// TIA Portal V17 export
// export: Created 2024-08-26T21:07:16.3751561Z, ExportSetting WithDefaults, DisplayName Totally Integrated Automation Portal, DisplayVersion V17 Update 7, DisplayName TIA Portal Openness, DisplayVersion V17 Update 7, DisplayName TIA Portal Version Control Interface, DisplayVersion V17, DisplayName SINAMICS Startdrive Advanced, DisplayVersion V17 SP2, DisplayName SINAMICS Startdrive G110M, G120, G120C, G120D, G120P, G115D, DisplayVersion V17 SP2, DisplayName SINAMICS Startdrive G130, G150, S120, S150, SINAMICS MV, S210, DisplayVersion V17 SP2, DisplayName STEP 7 Professional, DisplayVersion V17 Update 7, DisplayName STEP 7 Safety, DisplayVersion V17 Update 6, DisplayName WinCC Advanced / Unified PC, DisplayVersion V17 Update 7
FUNCTION "cylinderControl" : Void   // FC9, LAD
{ S7_Optimized_Access := 'TRUE' }
VERSION : 0.1
// stored: AutoNumber true, IsIECCheckEnabled false, SetENOAutomatically false, UDAEnableTagReadback false
   VAR_TEMP
      enableCylinders : Bool;
   END_VAR
   VAR_TEMP   // added for the SCL form of the ladder/FBD networks
      _w1 : Bool;
      _w2 : Bool;
   END_VAR
BEGIN

REGION Network 1
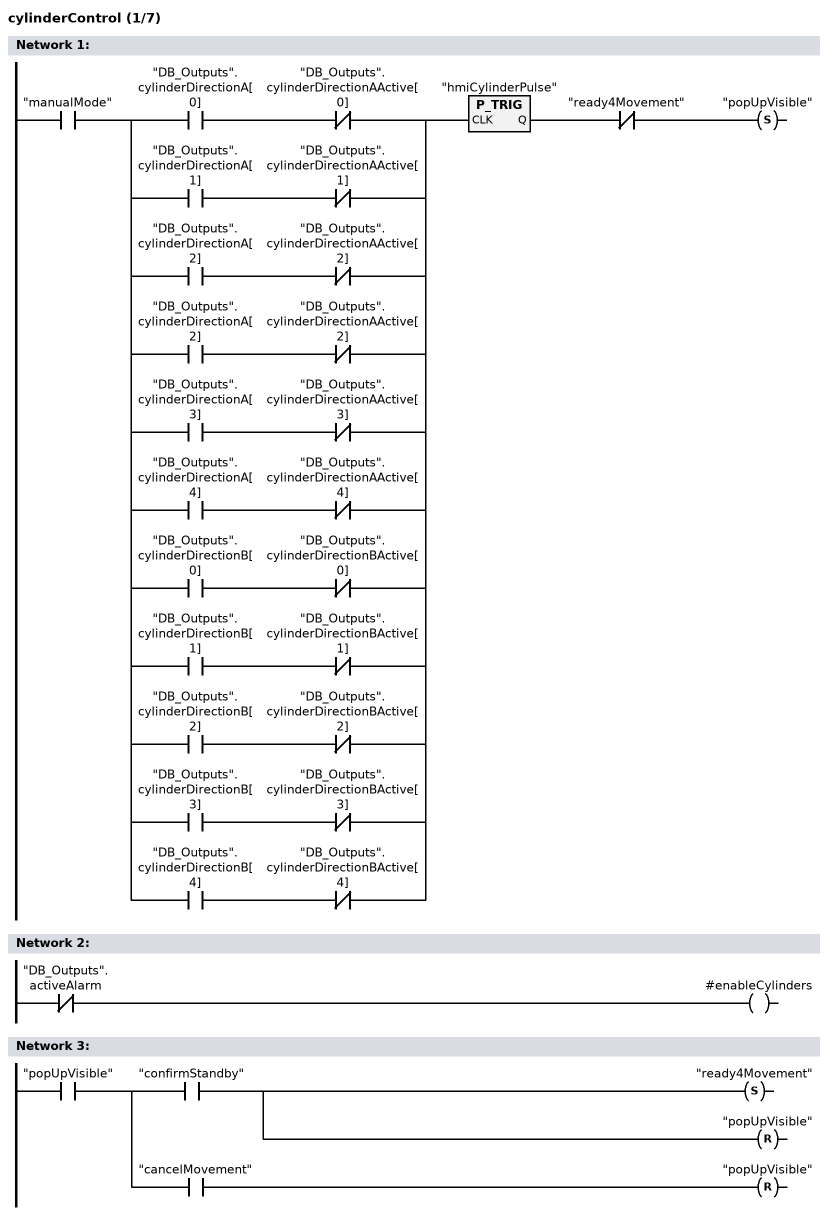
   RUNG wire#powerrail
      Contact( "manualMode" )
      wire#w1
      Contact( "DB_Outputs".cylinderDirectionA[0] )
      I_Contact( "DB_Outputs".cylinderDirectionAActive[0] )
      wire#w2
      P_Trig( "hmiCylinderPulse" )
      I_Contact( "ready4Movement" )
      S_Coil( "popUpVisible" )
   END_RUNG
   RUNG wire#w1
      Contact( "DB_Outputs".cylinderDirectionA[1] )
      I_Contact( "DB_Outputs".cylinderDirectionAActive[1] )
   END_RUNG wire#w2
   RUNG wire#w1
      Contact( "DB_Outputs".cylinderDirectionA[2] )
      I_Contact( "DB_Outputs".cylinderDirectionAActive[2] )
   END_RUNG wire#w2
   RUNG wire#w1
      Contact( "DB_Outputs".cylinderDirectionA[2] )
      I_Contact( "DB_Outputs".cylinderDirectionAActive[2] )
   END_RUNG wire#w2
   RUNG wire#w1
      Contact( "DB_Outputs".cylinderDirectionA[3] )
      I_Contact( "DB_Outputs".cylinderDirectionAActive[3] )
   END_RUNG wire#w2
   RUNG wire#w1
      Contact( "DB_Outputs".cylinderDirectionA[4] )
      I_Contact( "DB_Outputs".cylinderDirectionAActive[4] )
   END_RUNG wire#w2
   RUNG wire#w1
      Contact( "DB_Outputs".cylinderDirectionB[0] )
      I_Contact( "DB_Outputs".cylinderDirectionBActive[0] )
   END_RUNG wire#w2
   RUNG wire#w1
      Contact( "DB_Outputs".cylinderDirectionB[1] )
      I_Contact( "DB_Outputs".cylinderDirectionBActive[1] )
   END_RUNG wire#w2
   RUNG wire#w1
      Contact( "DB_Outputs".cylinderDirectionB[2] )
      I_Contact( "DB_Outputs".cylinderDirectionBActive[2] )
   END_RUNG wire#w2
   RUNG wire#w1
      Contact( "DB_Outputs".cylinderDirectionB[3] )
      I_Contact( "DB_Outputs".cylinderDirectionBActive[3] )
   END_RUNG wire#w2
   RUNG wire#w1
      Contact( "DB_Outputs".cylinderDirectionB[4] )
      I_Contact( "DB_Outputs".cylinderDirectionBActive[4] )
   END_RUNG wire#w2
   // the same network as SCL:
   #_w1 := "manualMode" AND (("DB_Outputs".cylinderDirectionA[0] AND NOT "DB_Outputs".cylinderDirectionAActive[0]) OR ("DB_Outputs".cylinderDirectionA[1] AND NOT "DB_Outputs".cylinderDirectionAActive[1]) OR ("DB_Outputs".cylinderDirectionA[2] AND NOT "DB_Outputs".cylinderDirectionAActive[2]) OR ("DB_Outputs".cylinderDirectionA[2] AND NOT "DB_Outputs".cylinderDirectionAActive[2]) OR ("DB_Outputs".cylinderDirectionA[3] AND NOT "DB_Outputs".cylinderDirectionAActive[3]) OR ("DB_Outputs".cylinderDirectionA[4] AND NOT "DB_Outputs".cylinderDirectionAActive[4]) OR ("DB_Outputs".cylinderDirectionB[0] AND NOT "DB_Outputs".cylinderDirectionBActive[0]) OR ("DB_Outputs".cylinderDirectionB[1] AND NOT "DB_Outputs".cylinderDirectionBActive[1]) OR ("DB_Outputs".cylinderDirectionB[2] AND NOT "DB_Outputs".cylinderDirectionBActive[2]) OR ("DB_Outputs".cylinderDirectionB[3] AND NOT "DB_Outputs".cylinderDirectionBActive[3]) OR ("DB_Outputs".cylinderDirectionB[4] AND NOT "DB_Outputs".cylinderDirectionBActive[4]));
   #_w2 := #_w1 AND NOT "hmiCylinderPulse";   // rising edge
   "hmiCylinderPulse" := #_w1;
   IF #_w2 AND NOT "ready4Movement" THEN "popUpVisible" := TRUE; END_IF;
END_REGION

REGION Network 2
   RUNG wire#powerrail
      I_Contact( "DB_Outputs".activeAlarm )
      Coil( #enableCylinders )
   END_RUNG
   // the same network as SCL:
   #enableCylinders := NOT "DB_Outputs".activeAlarm;
END_REGION

REGION Network 3
   RUNG wire#powerrail
      Contact( "popUpVisible" )
      wire#w1
      Contact( "confirmStandby" )
      wire#w2
      S_Coil( "ready4Movement" )
   END_RUNG
   RUNG wire#w2
      R_Coil( "popUpVisible" )
   END_RUNG
   RUNG wire#w1
      Contact( "cancelMovement" )
      R_Coil( "popUpVisible" )
   END_RUNG
   // the same network as SCL:
   IF "popUpVisible" AND "confirmStandby" THEN "ready4Movement" := TRUE; END_IF;
   #_w1 := "popUpVisible";
   IF "popUpVisible" AND "confirmStandby" THEN "popUpVisible" := FALSE; END_IF;
   IF #_w1 AND "cancelMovement" THEN "popUpVisible" := FALSE; END_IF;
END_REGION

REGION Network 4: EXT CYL 1.- LEFT TOOLING LOCK EXTENDED
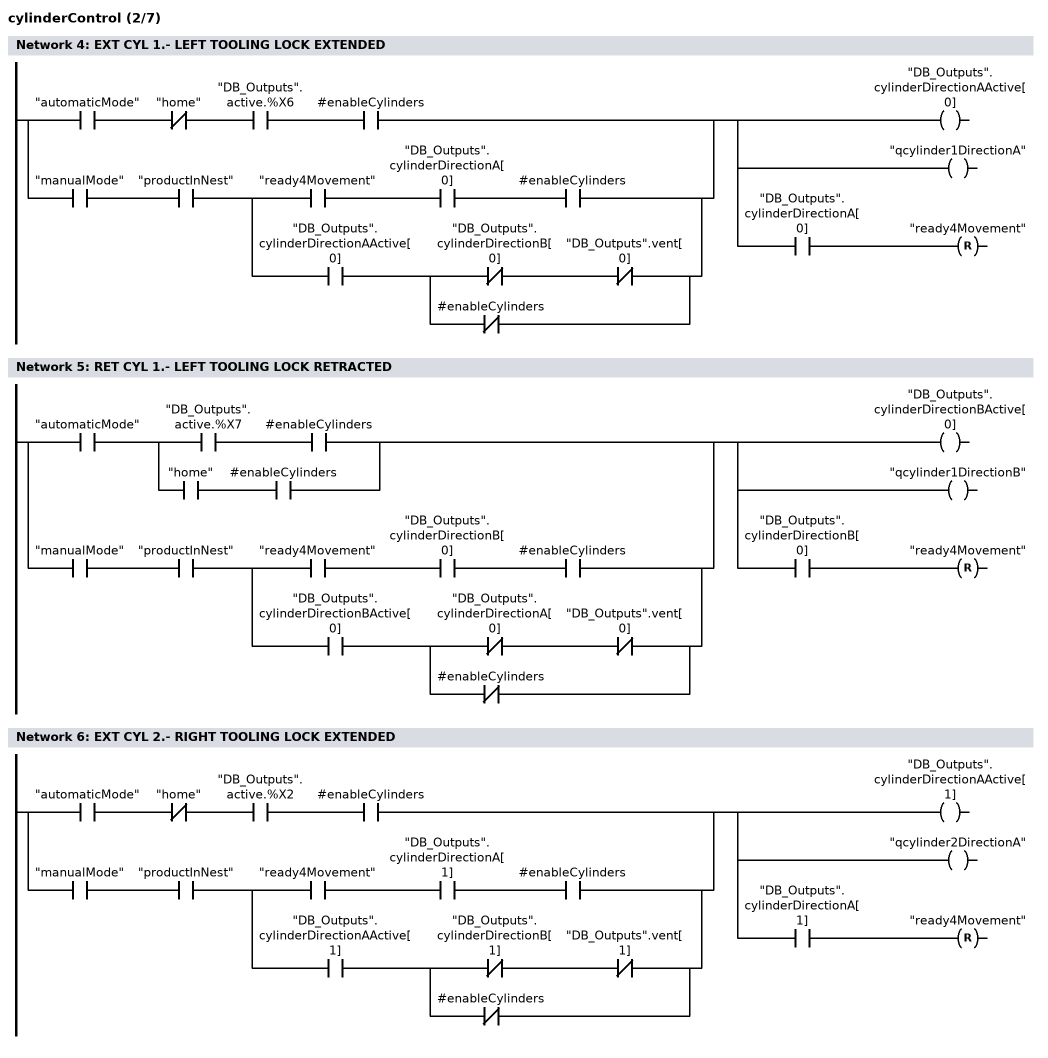
   RUNG wire#powerrail
      Contact( "automaticMode" )
      I_Contact( "home" )
      Contact( "DB_Outputs".active.%X6 )
      Contact( #enableCylinders )
      wire#w1
      Coil( "DB_Outputs".cylinderDirectionAActive[0] )
   END_RUNG
   RUNG wire#powerrail
      Contact( "manualMode" )
      Contact( "productInNest" )
      wire#w2
      Contact( "ready4Movement" )
      Contact( "DB_Outputs".cylinderDirectionA[0] )
      Contact( #enableCylinders )
   END_RUNG wire#w1
   RUNG wire#w2
      Contact( "DB_Outputs".cylinderDirectionAActive[0] )
      wire#w3
      I_Contact( "DB_Outputs".cylinderDirectionB[0] )
      I_Contact( "DB_Outputs".vent[0] )
   END_RUNG wire#w1
   RUNG wire#w3
      I_Contact( #enableCylinders )
   END_RUNG wire#w1
   RUNG wire#w1
      Coil( "qcylinder1DirectionA" )
   END_RUNG
   RUNG wire#w1
      Contact( "DB_Outputs".cylinderDirectionA[0] )
      R_Coil( "ready4Movement" )
   END_RUNG
   // the same network as SCL:
   #_w1 := ("automaticMode" AND NOT "home" AND "DB_Outputs".active.%X6 AND #enableCylinders) OR ("manualMode" AND "productInNest" AND (("ready4Movement" AND "DB_Outputs".cylinderDirectionA[0] AND #enableCylinders) OR ("DB_Outputs".cylinderDirectionAActive[0] AND ((NOT "DB_Outputs".cylinderDirectionB[0] AND NOT "DB_Outputs".vent[0]) OR NOT #enableCylinders))));
   "DB_Outputs".cylinderDirectionAActive[0] := ("automaticMode" AND NOT "home" AND "DB_Outputs".active.%X6 AND #enableCylinders) OR ("manualMode" AND "productInNest" AND (("ready4Movement" AND "DB_Outputs".cylinderDirectionA[0] AND #enableCylinders) OR ("DB_Outputs".cylinderDirectionAActive[0] AND ((NOT "DB_Outputs".cylinderDirectionB[0] AND NOT "DB_Outputs".vent[0]) OR NOT #enableCylinders))));
   "qcylinder1DirectionA" := #_w1;
   IF #_w1 AND "DB_Outputs".cylinderDirectionA[0] THEN "ready4Movement" := FALSE; END_IF;
END_REGION

REGION Network 5: RET CYL 1.- LEFT TOOLING LOCK RETRACTED
   RUNG wire#powerrail
      Contact( "automaticMode" )
      wire#w1
      Contact( "DB_Outputs".active.%X7 )
      Contact( #enableCylinders )
      wire#w2
      Coil( "DB_Outputs".cylinderDirectionBActive[0] )
   END_RUNG
   RUNG wire#w1
      Contact( "home" )
      Contact( #enableCylinders )
   END_RUNG wire#w2
   RUNG wire#powerrail
      Contact( "manualMode" )
      Contact( "productInNest" )
      wire#w3
      Contact( "ready4Movement" )
      Contact( "DB_Outputs".cylinderDirectionB[0] )
      Contact( #enableCylinders )
   END_RUNG wire#w2
   RUNG wire#w3
      Contact( "DB_Outputs".cylinderDirectionBActive[0] )
      wire#w4
      I_Contact( "DB_Outputs".cylinderDirectionA[0] )
      I_Contact( "DB_Outputs".vent[0] )
   END_RUNG wire#w2
   RUNG wire#w4
      I_Contact( #enableCylinders )
   END_RUNG wire#w2
   RUNG wire#w2
      Coil( "qcylinder1DirectionB" )
   END_RUNG
   RUNG wire#w2
      Contact( "DB_Outputs".cylinderDirectionB[0] )
      R_Coil( "ready4Movement" )
   END_RUNG
   // the same network as SCL:
   #_w1 := ("automaticMode" AND (("DB_Outputs".active.%X7 AND #enableCylinders) OR ("home" AND #enableCylinders))) OR ("manualMode" AND "productInNest" AND (("ready4Movement" AND "DB_Outputs".cylinderDirectionB[0] AND #enableCylinders) OR ("DB_Outputs".cylinderDirectionBActive[0] AND ((NOT "DB_Outputs".cylinderDirectionA[0] AND NOT "DB_Outputs".vent[0]) OR NOT #enableCylinders))));
   "DB_Outputs".cylinderDirectionBActive[0] := ("automaticMode" AND (("DB_Outputs".active.%X7 AND #enableCylinders) OR ("home" AND #enableCylinders))) OR ("manualMode" AND "productInNest" AND (("ready4Movement" AND "DB_Outputs".cylinderDirectionB[0] AND #enableCylinders) OR ("DB_Outputs".cylinderDirectionBActive[0] AND ((NOT "DB_Outputs".cylinderDirectionA[0] AND NOT "DB_Outputs".vent[0]) OR NOT #enableCylinders))));
   "qcylinder1DirectionB" := #_w1;
   IF #_w1 AND "DB_Outputs".cylinderDirectionB[0] THEN "ready4Movement" := FALSE; END_IF;
END_REGION

REGION Network 6: EXT CYL 2.- RIGHT TOOLING LOCK EXTENDED
   RUNG wire#powerrail
      Contact( "automaticMode" )
      I_Contact( "home" )
      Contact( "DB_Outputs".active.%X2 )
      Contact( #enableCylinders )
      wire#w1
      Coil( "DB_Outputs".cylinderDirectionAActive[1] )
   END_RUNG
   RUNG wire#powerrail
      Contact( "manualMode" )
      Contact( "productInNest" )
      wire#w2
      Contact( "ready4Movement" )
      Contact( "DB_Outputs".cylinderDirectionA[1] )
      Contact( #enableCylinders )
   END_RUNG wire#w1
   RUNG wire#w2
      Contact( "DB_Outputs".cylinderDirectionAActive[1] )
      wire#w3
      I_Contact( "DB_Outputs".cylinderDirectionB[1] )
      I_Contact( "DB_Outputs".vent[1] )
   END_RUNG wire#w1
   RUNG wire#w3
      I_Contact( #enableCylinders )
   END_RUNG wire#w1
   RUNG wire#w1
      Coil( "qcylinder2DirectionA" )
   END_RUNG
   RUNG wire#w1
      Contact( "DB_Outputs".cylinderDirectionA[1] )
      R_Coil( "ready4Movement" )
   END_RUNG
   // the same network as SCL:
   #_w1 := ("automaticMode" AND NOT "home" AND "DB_Outputs".active.%X2 AND #enableCylinders) OR ("manualMode" AND "productInNest" AND (("ready4Movement" AND "DB_Outputs".cylinderDirectionA[1] AND #enableCylinders) OR ("DB_Outputs".cylinderDirectionAActive[1] AND ((NOT "DB_Outputs".cylinderDirectionB[1] AND NOT "DB_Outputs".vent[1]) OR NOT #enableCylinders))));
   "DB_Outputs".cylinderDirectionAActive[1] := ("automaticMode" AND NOT "home" AND "DB_Outputs".active.%X2 AND #enableCylinders) OR ("manualMode" AND "productInNest" AND (("ready4Movement" AND "DB_Outputs".cylinderDirectionA[1] AND #enableCylinders) OR ("DB_Outputs".cylinderDirectionAActive[1] AND ((NOT "DB_Outputs".cylinderDirectionB[1] AND NOT "DB_Outputs".vent[1]) OR NOT #enableCylinders))));
   "qcylinder2DirectionA" := #_w1;
   IF #_w1 AND "DB_Outputs".cylinderDirectionA[1] THEN "ready4Movement" := FALSE; END_IF;
END_REGION

REGION Network 7: RET CYL 2.- RIGHT TOOLING LOCK RETRACTED
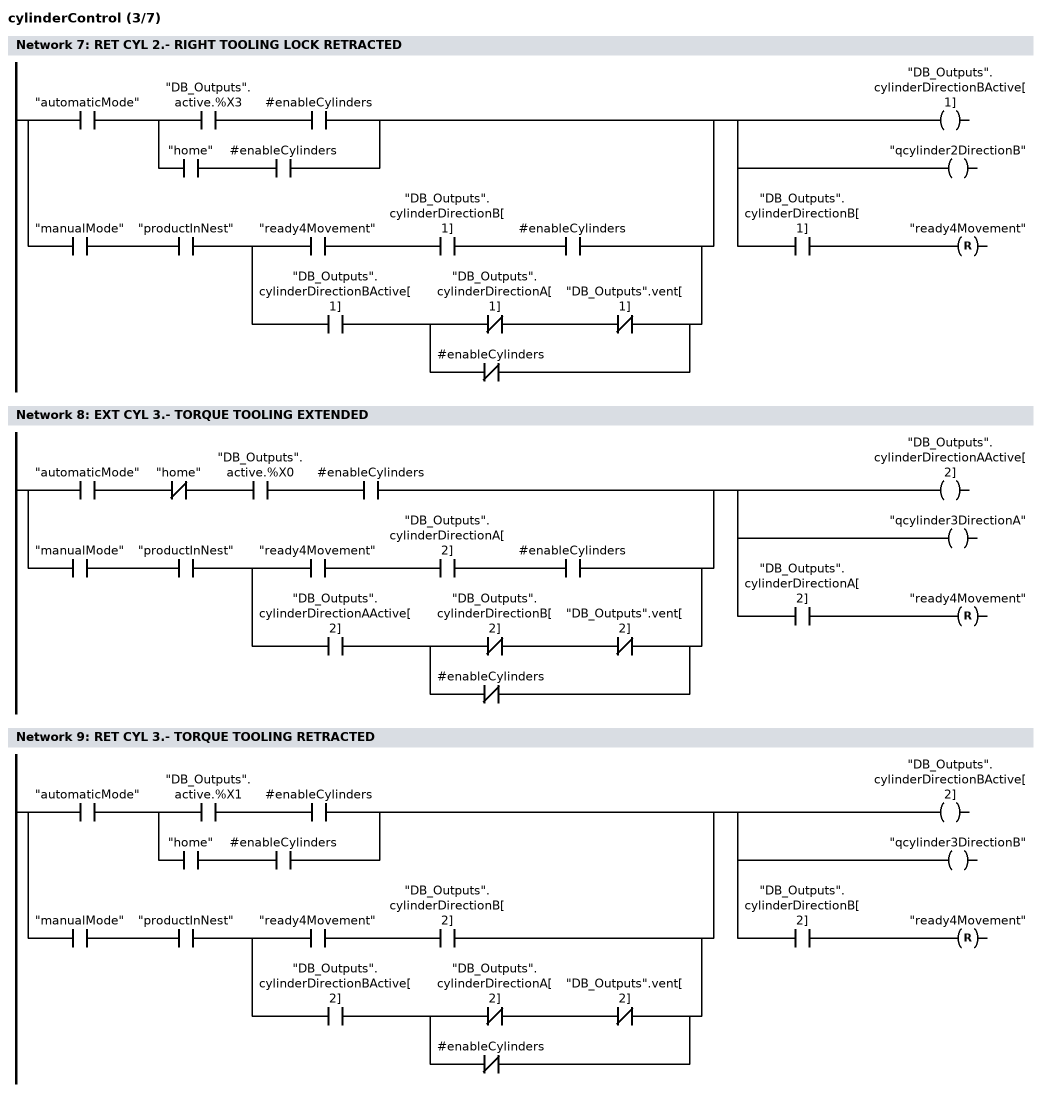
   RUNG wire#powerrail
      Contact( "automaticMode" )
      wire#w1
      Contact( "DB_Outputs".active.%X3 )
      Contact( #enableCylinders )
      wire#w2
      Coil( "DB_Outputs".cylinderDirectionBActive[1] )
   END_RUNG
   RUNG wire#w1
      Contact( "home" )
      Contact( #enableCylinders )
   END_RUNG wire#w2
   RUNG wire#powerrail
      Contact( "manualMode" )
      Contact( "productInNest" )
      wire#w3
      Contact( "ready4Movement" )
      Contact( "DB_Outputs".cylinderDirectionB[1] )
      Contact( #enableCylinders )
   END_RUNG wire#w2
   RUNG wire#w3
      Contact( "DB_Outputs".cylinderDirectionBActive[1] )
      wire#w4
      I_Contact( "DB_Outputs".cylinderDirectionA[1] )
      I_Contact( "DB_Outputs".vent[1] )
   END_RUNG wire#w2
   RUNG wire#w4
      I_Contact( #enableCylinders )
   END_RUNG wire#w2
   RUNG wire#w2
      Coil( "qcylinder2DirectionB" )
   END_RUNG
   RUNG wire#w2
      Contact( "DB_Outputs".cylinderDirectionB[1] )
      R_Coil( "ready4Movement" )
   END_RUNG
   // the same network as SCL:
   #_w1 := ("automaticMode" AND (("DB_Outputs".active.%X3 AND #enableCylinders) OR ("home" AND #enableCylinders))) OR ("manualMode" AND "productInNest" AND (("ready4Movement" AND "DB_Outputs".cylinderDirectionB[1] AND #enableCylinders) OR ("DB_Outputs".cylinderDirectionBActive[1] AND ((NOT "DB_Outputs".cylinderDirectionA[1] AND NOT "DB_Outputs".vent[1]) OR NOT #enableCylinders))));
   "DB_Outputs".cylinderDirectionBActive[1] := ("automaticMode" AND (("DB_Outputs".active.%X3 AND #enableCylinders) OR ("home" AND #enableCylinders))) OR ("manualMode" AND "productInNest" AND (("ready4Movement" AND "DB_Outputs".cylinderDirectionB[1] AND #enableCylinders) OR ("DB_Outputs".cylinderDirectionBActive[1] AND ((NOT "DB_Outputs".cylinderDirectionA[1] AND NOT "DB_Outputs".vent[1]) OR NOT #enableCylinders))));
   "qcylinder2DirectionB" := #_w1;
   IF #_w1 AND "DB_Outputs".cylinderDirectionB[1] THEN "ready4Movement" := FALSE; END_IF;
END_REGION

REGION Network 8: EXT CYL 3.- TORQUE TOOLING EXTENDED
   RUNG wire#powerrail
      Contact( "automaticMode" )
      I_Contact( "home" )
      Contact( "DB_Outputs".active.%X0 )
      Contact( #enableCylinders )
      wire#w1
      Coil( "DB_Outputs".cylinderDirectionAActive[2] )
   END_RUNG
   RUNG wire#powerrail
      Contact( "manualMode" )
      Contact( "productInNest" )
      wire#w2
      Contact( "ready4Movement" )
      Contact( "DB_Outputs".cylinderDirectionA[2] )
      Contact( #enableCylinders )
   END_RUNG wire#w1
   RUNG wire#w2
      Contact( "DB_Outputs".cylinderDirectionAActive[2] )
      wire#w3
      I_Contact( "DB_Outputs".cylinderDirectionB[2] )
      I_Contact( "DB_Outputs".vent[2] )
   END_RUNG wire#w1
   RUNG wire#w3
      I_Contact( #enableCylinders )
   END_RUNG wire#w1
   RUNG wire#w1
      Coil( "qcylinder3DirectionA" )
   END_RUNG
   RUNG wire#w1
      Contact( "DB_Outputs".cylinderDirectionA[2] )
      R_Coil( "ready4Movement" )
   END_RUNG
   // the same network as SCL:
   #_w1 := ("automaticMode" AND NOT "home" AND "DB_Outputs".active.%X0 AND #enableCylinders) OR ("manualMode" AND "productInNest" AND (("ready4Movement" AND "DB_Outputs".cylinderDirectionA[2] AND #enableCylinders) OR ("DB_Outputs".cylinderDirectionAActive[2] AND ((NOT "DB_Outputs".cylinderDirectionB[2] AND NOT "DB_Outputs".vent[2]) OR NOT #enableCylinders))));
   "DB_Outputs".cylinderDirectionAActive[2] := ("automaticMode" AND NOT "home" AND "DB_Outputs".active.%X0 AND #enableCylinders) OR ("manualMode" AND "productInNest" AND (("ready4Movement" AND "DB_Outputs".cylinderDirectionA[2] AND #enableCylinders) OR ("DB_Outputs".cylinderDirectionAActive[2] AND ((NOT "DB_Outputs".cylinderDirectionB[2] AND NOT "DB_Outputs".vent[2]) OR NOT #enableCylinders))));
   "qcylinder3DirectionA" := #_w1;
   IF #_w1 AND "DB_Outputs".cylinderDirectionA[2] THEN "ready4Movement" := FALSE; END_IF;
END_REGION

REGION Network 9: RET CYL 3.- TORQUE TOOLING RETRACTED
   RUNG wire#powerrail
      Contact( "automaticMode" )
      wire#w1
      Contact( "DB_Outputs".active.%X1 )
      Contact( #enableCylinders )
      wire#w2
      Coil( "DB_Outputs".cylinderDirectionBActive[2] )
   END_RUNG
   RUNG wire#w1
      Contact( "home" )
      Contact( #enableCylinders )
   END_RUNG wire#w2
   RUNG wire#powerrail
      Contact( "manualMode" )
      Contact( "productInNest" )
      wire#w3
      Contact( "ready4Movement" )
      Contact( "DB_Outputs".cylinderDirectionB[2] )
   END_RUNG wire#w2
   RUNG wire#w3
      Contact( "DB_Outputs".cylinderDirectionBActive[2] )
      wire#w4
      I_Contact( "DB_Outputs".cylinderDirectionA[2] )
      I_Contact( "DB_Outputs".vent[2] )
   END_RUNG wire#w2
   RUNG wire#w4
      I_Contact( #enableCylinders )
   END_RUNG wire#w2
   RUNG wire#w2
      Coil( "qcylinder3DirectionB" )
   END_RUNG
   RUNG wire#w2
      Contact( "DB_Outputs".cylinderDirectionB[2] )
      R_Coil( "ready4Movement" )
   END_RUNG
   // the same network as SCL:
   #_w1 := ("automaticMode" AND (("DB_Outputs".active.%X1 AND #enableCylinders) OR ("home" AND #enableCylinders))) OR ("manualMode" AND "productInNest" AND (("ready4Movement" AND "DB_Outputs".cylinderDirectionB[2]) OR ("DB_Outputs".cylinderDirectionBActive[2] AND ((NOT "DB_Outputs".cylinderDirectionA[2] AND NOT "DB_Outputs".vent[2]) OR NOT #enableCylinders))));
   "DB_Outputs".cylinderDirectionBActive[2] := ("automaticMode" AND (("DB_Outputs".active.%X1 AND #enableCylinders) OR ("home" AND #enableCylinders))) OR ("manualMode" AND "productInNest" AND (("ready4Movement" AND "DB_Outputs".cylinderDirectionB[2]) OR ("DB_Outputs".cylinderDirectionBActive[2] AND ((NOT "DB_Outputs".cylinderDirectionA[2] AND NOT "DB_Outputs".vent[2]) OR NOT #enableCylinders))));
   "qcylinder3DirectionB" := #_w1;
   IF #_w1 AND "DB_Outputs".cylinderDirectionB[2] THEN "ready4Movement" := FALSE; END_IF;
END_REGION

REGION Network 10: EXT CYL 4.- RIGTH ROD INSERTION EXTENDED
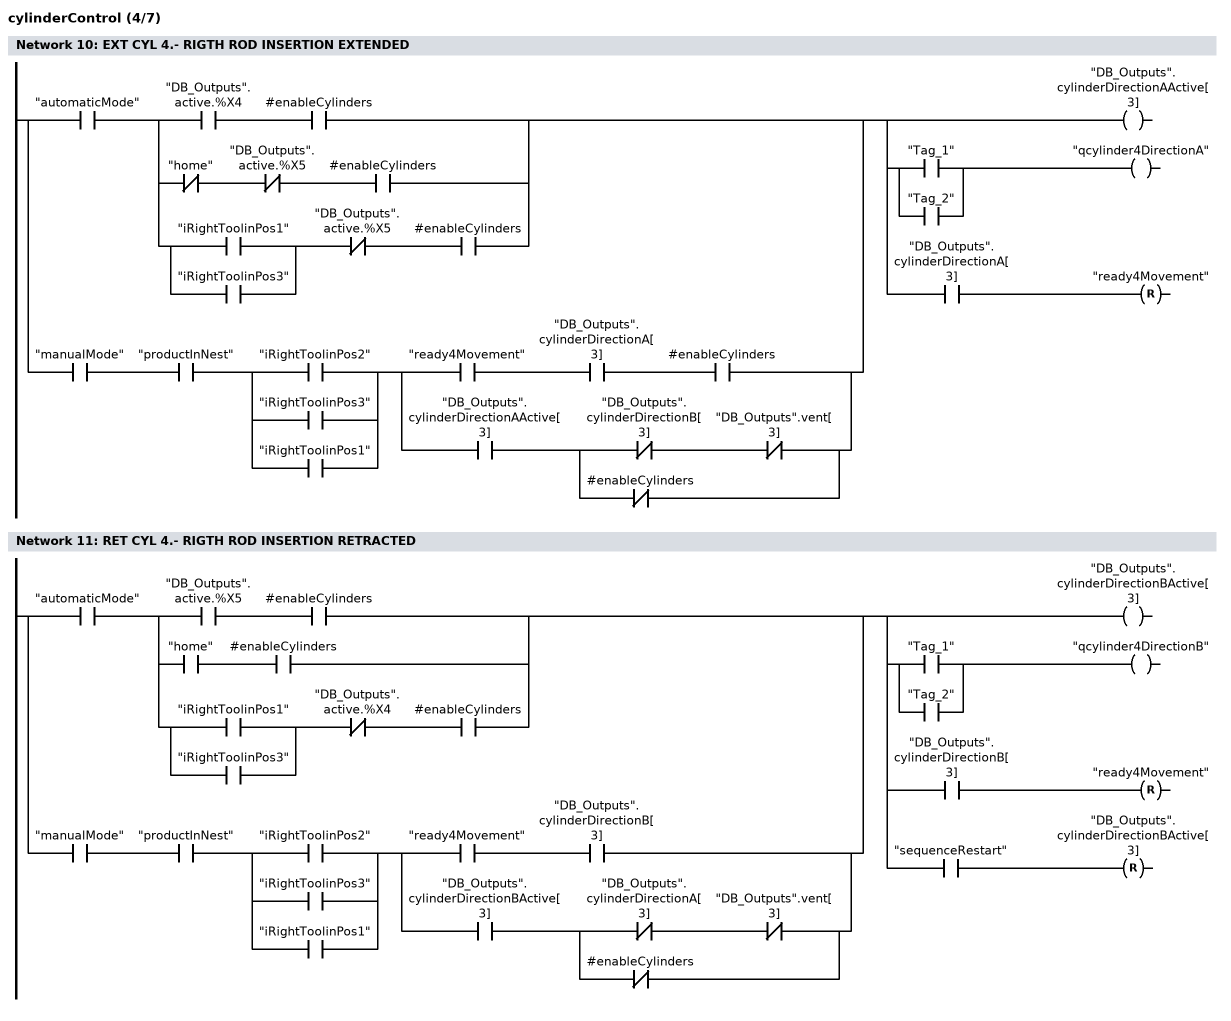
   RUNG wire#powerrail
      Contact( "automaticMode" )
      wire#w1
      Contact( "DB_Outputs".active.%X4 )
      Contact( #enableCylinders )
      wire#w2
      Coil( "DB_Outputs".cylinderDirectionAActive[3] )
   END_RUNG
   RUNG wire#w1
      I_Contact( "home" )
      I_Contact( "DB_Outputs".active.%X5 )
      Contact( #enableCylinders )
   END_RUNG wire#w2
   RUNG wire#w1
      Contact( "iRightToolinPos1" )
      wire#w3
      I_Contact( "DB_Outputs".active.%X5 )
      Contact( #enableCylinders )
   END_RUNG wire#w2
   RUNG wire#w1
      Contact( "iRightToolinPos3" )
   END_RUNG wire#w3
   RUNG wire#powerrail
      Contact( "manualMode" )
      Contact( "productInNest" )
      wire#w4
      Contact( "iRightToolinPos2" )
      wire#w5
      Contact( "ready4Movement" )
      Contact( "DB_Outputs".cylinderDirectionA[3] )
      Contact( #enableCylinders )
   END_RUNG wire#w2
   RUNG wire#w4
      Contact( "iRightToolinPos3" )
   END_RUNG wire#w5
   RUNG wire#w4
      Contact( "iRightToolinPos1" )
   END_RUNG wire#w5
   RUNG wire#w5
      Contact( "DB_Outputs".cylinderDirectionAActive[3] )
      wire#w6
      I_Contact( "DB_Outputs".cylinderDirectionB[3] )
      I_Contact( "DB_Outputs".vent[3] )
   END_RUNG wire#w2
   RUNG wire#w6
      I_Contact( #enableCylinders )
   END_RUNG wire#w2
   RUNG wire#w2
      Contact( "Tag_1" )
      wire#w7
      Coil( "qcylinder4DirectionA" )
   END_RUNG
   RUNG wire#w2
      Contact( "Tag_2" )
   END_RUNG wire#w7
   RUNG wire#w2
      Contact( "DB_Outputs".cylinderDirectionA[3] )
      R_Coil( "ready4Movement" )
   END_RUNG
   // the same network as SCL:
   #_w1 := ("automaticMode" AND (("DB_Outputs".active.%X4 AND #enableCylinders) OR (NOT "home" AND NOT "DB_Outputs".active.%X5 AND #enableCylinders) OR (("iRightToolinPos1" OR "iRightToolinPos3") AND NOT "DB_Outputs".active.%X5 AND #enableCylinders))) OR ("manualMode" AND "productInNest" AND ("iRightToolinPos2" OR "iRightToolinPos3" OR "iRightToolinPos1") AND (("ready4Movement" AND "DB_Outputs".cylinderDirectionA[3] AND #enableCylinders) OR ("DB_Outputs".cylinderDirectionAActive[3] AND ((NOT "DB_Outputs".cylinderDirectionB[3] AND NOT "DB_Outputs".vent[3]) OR NOT #enableCylinders))));
   "DB_Outputs".cylinderDirectionAActive[3] := ("automaticMode" AND (("DB_Outputs".active.%X4 AND #enableCylinders) OR (NOT "home" AND NOT "DB_Outputs".active.%X5 AND #enableCylinders) OR (("iRightToolinPos1" OR "iRightToolinPos3") AND NOT "DB_Outputs".active.%X5 AND #enableCylinders))) OR ("manualMode" AND "productInNest" AND ("iRightToolinPos2" OR "iRightToolinPos3" OR "iRightToolinPos1") AND (("ready4Movement" AND "DB_Outputs".cylinderDirectionA[3] AND #enableCylinders) OR ("DB_Outputs".cylinderDirectionAActive[3] AND ((NOT "DB_Outputs".cylinderDirectionB[3] AND NOT "DB_Outputs".vent[3]) OR NOT #enableCylinders))));
   "qcylinder4DirectionA" := #_w1 AND ("Tag_1" OR "Tag_2");
   IF #_w1 AND "DB_Outputs".cylinderDirectionA[3] THEN "ready4Movement" := FALSE; END_IF;
END_REGION

REGION Network 11: RET CYL 4.- RIGTH ROD INSERTION RETRACTED
   RUNG wire#powerrail
      Contact( "automaticMode" )
      wire#w1
      Contact( "DB_Outputs".active.%X5 )
      Contact( #enableCylinders )
      wire#w2
      Coil( "DB_Outputs".cylinderDirectionBActive[3] )
   END_RUNG
   RUNG wire#w1
      Contact( "home" )
      Contact( #enableCylinders )
   END_RUNG wire#w2
   RUNG wire#w1
      Contact( "iRightToolinPos1" )
      wire#w3
      I_Contact( "DB_Outputs".active.%X4 )
      Contact( #enableCylinders )
   END_RUNG wire#w2
   RUNG wire#w1
      Contact( "iRightToolinPos3" )
   END_RUNG wire#w3
   RUNG wire#powerrail
      Contact( "manualMode" )
      Contact( "productInNest" )
      wire#w4
      Contact( "iRightToolinPos2" )
      wire#w5
      Contact( "ready4Movement" )
      Contact( "DB_Outputs".cylinderDirectionB[3] )
   END_RUNG wire#w2
   RUNG wire#w4
      Contact( "iRightToolinPos3" )
   END_RUNG wire#w5
   RUNG wire#w4
      Contact( "iRightToolinPos1" )
   END_RUNG wire#w5
   RUNG wire#w5
      Contact( "DB_Outputs".cylinderDirectionBActive[3] )
      wire#w6
      I_Contact( "DB_Outputs".cylinderDirectionA[3] )
      I_Contact( "DB_Outputs".vent[3] )
   END_RUNG wire#w2
   RUNG wire#w6
      I_Contact( #enableCylinders )
   END_RUNG wire#w2
   RUNG wire#w2
      Contact( "Tag_1" )
      wire#w7
      Coil( "qcylinder4DirectionB" )
   END_RUNG
   RUNG wire#w2
      Contact( "Tag_2" )
   END_RUNG wire#w7
   RUNG wire#w2
      Contact( "DB_Outputs".cylinderDirectionB[3] )
      R_Coil( "ready4Movement" )
   END_RUNG
   RUNG wire#w2
      Contact( "sequenceRestart" )
      R_Coil( "DB_Outputs".cylinderDirectionBActive[3] )
   END_RUNG
   // the same network as SCL:
   #_w1 := ("automaticMode" AND (("DB_Outputs".active.%X5 AND #enableCylinders) OR ("home" AND #enableCylinders) OR (("iRightToolinPos1" OR "iRightToolinPos3") AND NOT "DB_Outputs".active.%X4 AND #enableCylinders))) OR ("manualMode" AND "productInNest" AND ("iRightToolinPos2" OR "iRightToolinPos3" OR "iRightToolinPos1") AND (("ready4Movement" AND "DB_Outputs".cylinderDirectionB[3]) OR ("DB_Outputs".cylinderDirectionBActive[3] AND ((NOT "DB_Outputs".cylinderDirectionA[3] AND NOT "DB_Outputs".vent[3]) OR NOT #enableCylinders))));
   "DB_Outputs".cylinderDirectionBActive[3] := ("automaticMode" AND (("DB_Outputs".active.%X5 AND #enableCylinders) OR ("home" AND #enableCylinders) OR (("iRightToolinPos1" OR "iRightToolinPos3") AND NOT "DB_Outputs".active.%X4 AND #enableCylinders))) OR ("manualMode" AND "productInNest" AND ("iRightToolinPos2" OR "iRightToolinPos3" OR "iRightToolinPos1") AND (("ready4Movement" AND "DB_Outputs".cylinderDirectionB[3]) OR ("DB_Outputs".cylinderDirectionBActive[3] AND ((NOT "DB_Outputs".cylinderDirectionA[3] AND NOT "DB_Outputs".vent[3]) OR NOT #enableCylinders))));
   "qcylinder4DirectionB" := #_w1 AND ("Tag_1" OR "Tag_2");
   IF #_w1 AND "DB_Outputs".cylinderDirectionB[3] THEN "ready4Movement" := FALSE; END_IF;
   IF #_w1 AND "sequenceRestart" THEN "DB_Outputs".cylinderDirectionBActive[3] := FALSE; END_IF;
END_REGION

REGION Network 12: EXT CYL 5.- LEFT WASHER/ROD INSERTION EXTENDED
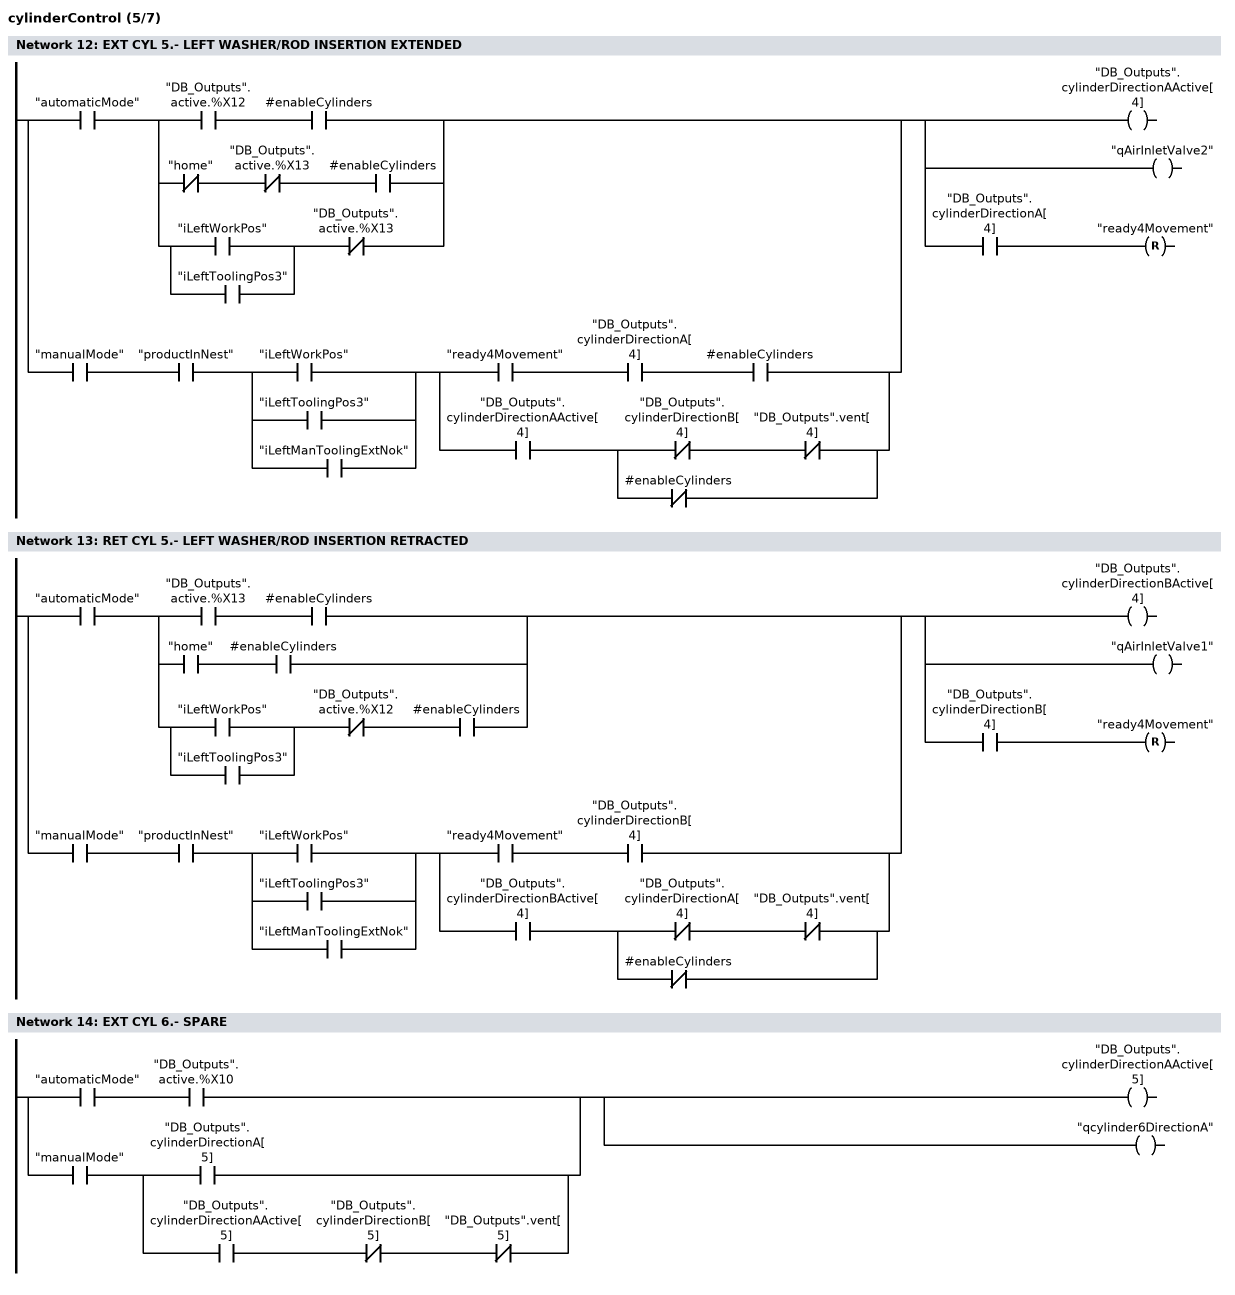
   RUNG wire#powerrail
      Contact( "automaticMode" )
      wire#w1
      Contact( "DB_Outputs".active.%X12 )
      Contact( #enableCylinders )
      wire#w2
      Coil( "DB_Outputs".cylinderDirectionAActive[4] )
   END_RUNG
   RUNG wire#w1
      I_Contact( "home" )
      I_Contact( "DB_Outputs".active.%X13 )
      Contact( #enableCylinders )
   END_RUNG wire#w2
   RUNG wire#w1
      Contact( "iLeftWorkPos" )
      wire#w3
      I_Contact( "DB_Outputs".active.%X13 )
   END_RUNG wire#w2
   RUNG wire#w1
      Contact( "iLeftToolingPos3" )
   END_RUNG wire#w3
   RUNG wire#powerrail
      Contact( "manualMode" )
      Contact( "productInNest" )
      wire#w4
      Contact( "iLeftWorkPos" )
      wire#w5
      Contact( "ready4Movement" )
      Contact( "DB_Outputs".cylinderDirectionA[4] )
      Contact( #enableCylinders )
   END_RUNG wire#w2
   RUNG wire#w4
      Contact( "iLeftToolingPos3" )
   END_RUNG wire#w5
   RUNG wire#w4
      Contact( "iLeftManToolingExtNok" )
   END_RUNG wire#w5
   RUNG wire#w5
      Contact( "DB_Outputs".cylinderDirectionAActive[4] )
      wire#w6
      I_Contact( "DB_Outputs".cylinderDirectionB[4] )
      I_Contact( "DB_Outputs".vent[4] )
   END_RUNG wire#w2
   RUNG wire#w6
      I_Contact( #enableCylinders )
   END_RUNG wire#w2
   RUNG wire#w2
      Coil( "qAirInletValve2" )
   END_RUNG
   RUNG wire#w2
      Contact( "DB_Outputs".cylinderDirectionA[4] )
      R_Coil( "ready4Movement" )
   END_RUNG
   // the same network as SCL:
   #_w1 := ("automaticMode" AND (("DB_Outputs".active.%X12 AND #enableCylinders) OR (NOT "home" AND NOT "DB_Outputs".active.%X13 AND #enableCylinders) OR (("iLeftWorkPos" OR "iLeftToolingPos3") AND NOT "DB_Outputs".active.%X13))) OR ("manualMode" AND "productInNest" AND ("iLeftWorkPos" OR "iLeftToolingPos3" OR "iLeftManToolingExtNok") AND (("ready4Movement" AND "DB_Outputs".cylinderDirectionA[4] AND #enableCylinders) OR ("DB_Outputs".cylinderDirectionAActive[4] AND ((NOT "DB_Outputs".cylinderDirectionB[4] AND NOT "DB_Outputs".vent[4]) OR NOT #enableCylinders))));
   "DB_Outputs".cylinderDirectionAActive[4] := ("automaticMode" AND (("DB_Outputs".active.%X12 AND #enableCylinders) OR (NOT "home" AND NOT "DB_Outputs".active.%X13 AND #enableCylinders) OR (("iLeftWorkPos" OR "iLeftToolingPos3") AND NOT "DB_Outputs".active.%X13))) OR ("manualMode" AND "productInNest" AND ("iLeftWorkPos" OR "iLeftToolingPos3" OR "iLeftManToolingExtNok") AND (("ready4Movement" AND "DB_Outputs".cylinderDirectionA[4] AND #enableCylinders) OR ("DB_Outputs".cylinderDirectionAActive[4] AND ((NOT "DB_Outputs".cylinderDirectionB[4] AND NOT "DB_Outputs".vent[4]) OR NOT #enableCylinders))));
   "qAirInletValve2" := #_w1;
   IF #_w1 AND "DB_Outputs".cylinderDirectionA[4] THEN "ready4Movement" := FALSE; END_IF;
END_REGION

REGION Network 13: RET CYL 5.- LEFT WASHER/ROD INSERTION RETRACTED
   RUNG wire#powerrail
      Contact( "automaticMode" )
      wire#w1
      Contact( "DB_Outputs".active.%X13 )
      Contact( #enableCylinders )
      wire#w2
      Coil( "DB_Outputs".cylinderDirectionBActive[4] )
   END_RUNG
   RUNG wire#w1
      Contact( "home" )
      Contact( #enableCylinders )
   END_RUNG wire#w2
   RUNG wire#w1
      Contact( "iLeftWorkPos" )
      wire#w3
      I_Contact( "DB_Outputs".active.%X12 )
      Contact( #enableCylinders )
   END_RUNG wire#w2
   RUNG wire#w1
      Contact( "iLeftToolingPos3" )
   END_RUNG wire#w3
   RUNG wire#powerrail
      Contact( "manualMode" )
      Contact( "productInNest" )
      wire#w4
      Contact( "iLeftWorkPos" )
      wire#w5
      Contact( "ready4Movement" )
      Contact( "DB_Outputs".cylinderDirectionB[4] )
   END_RUNG wire#w2
   RUNG wire#w4
      Contact( "iLeftToolingPos3" )
   END_RUNG wire#w5
   RUNG wire#w4
      Contact( "iLeftManToolingExtNok" )
   END_RUNG wire#w5
   RUNG wire#w5
      Contact( "DB_Outputs".cylinderDirectionBActive[4] )
      wire#w6
      I_Contact( "DB_Outputs".cylinderDirectionA[4] )
      I_Contact( "DB_Outputs".vent[4] )
   END_RUNG wire#w2
   RUNG wire#w6
      I_Contact( #enableCylinders )
   END_RUNG wire#w2
   RUNG wire#w2
      Coil( "qAirInletValve1" )
   END_RUNG
   RUNG wire#w2
      Contact( "DB_Outputs".cylinderDirectionB[4] )
      R_Coil( "ready4Movement" )
   END_RUNG
   // the same network as SCL:
   #_w1 := ("automaticMode" AND (("DB_Outputs".active.%X13 AND #enableCylinders) OR ("home" AND #enableCylinders) OR (("iLeftWorkPos" OR "iLeftToolingPos3") AND NOT "DB_Outputs".active.%X12 AND #enableCylinders))) OR ("manualMode" AND "productInNest" AND ("iLeftWorkPos" OR "iLeftToolingPos3" OR "iLeftManToolingExtNok") AND (("ready4Movement" AND "DB_Outputs".cylinderDirectionB[4]) OR ("DB_Outputs".cylinderDirectionBActive[4] AND ((NOT "DB_Outputs".cylinderDirectionA[4] AND NOT "DB_Outputs".vent[4]) OR NOT #enableCylinders))));
   "DB_Outputs".cylinderDirectionBActive[4] := ("automaticMode" AND (("DB_Outputs".active.%X13 AND #enableCylinders) OR ("home" AND #enableCylinders) OR (("iLeftWorkPos" OR "iLeftToolingPos3") AND NOT "DB_Outputs".active.%X12 AND #enableCylinders))) OR ("manualMode" AND "productInNest" AND ("iLeftWorkPos" OR "iLeftToolingPos3" OR "iLeftManToolingExtNok") AND (("ready4Movement" AND "DB_Outputs".cylinderDirectionB[4]) OR ("DB_Outputs".cylinderDirectionBActive[4] AND ((NOT "DB_Outputs".cylinderDirectionA[4] AND NOT "DB_Outputs".vent[4]) OR NOT #enableCylinders))));
   "qAirInletValve1" := #_w1;
   IF #_w1 AND "DB_Outputs".cylinderDirectionB[4] THEN "ready4Movement" := FALSE; END_IF;
END_REGION

REGION Network 14: EXT CYL 6.- SPARE
   RUNG wire#powerrail
      Contact( "automaticMode" )
      Contact( "DB_Outputs".active.%X10 )
      wire#w1
      Coil( "DB_Outputs".cylinderDirectionAActive[5] )
   END_RUNG
   RUNG wire#powerrail
      Contact( "manualMode" )
      wire#w2
      Contact( "DB_Outputs".cylinderDirectionA[5] )
   END_RUNG wire#w1
   RUNG wire#w2
      Contact( "DB_Outputs".cylinderDirectionAActive[5] )
      I_Contact( "DB_Outputs".cylinderDirectionB[5] )
      I_Contact( "DB_Outputs".vent[5] )
   END_RUNG wire#w1
   RUNG wire#w1
      Coil( "qcylinder6DirectionA" )
   END_RUNG
   // the same network as SCL:
   #_w1 := ("automaticMode" AND "DB_Outputs".active.%X10) OR ("manualMode" AND ("DB_Outputs".cylinderDirectionA[5] OR ("DB_Outputs".cylinderDirectionAActive[5] AND NOT "DB_Outputs".cylinderDirectionB[5] AND NOT "DB_Outputs".vent[5])));
   "DB_Outputs".cylinderDirectionAActive[5] := ("automaticMode" AND "DB_Outputs".active.%X10) OR ("manualMode" AND ("DB_Outputs".cylinderDirectionA[5] OR ("DB_Outputs".cylinderDirectionAActive[5] AND NOT "DB_Outputs".cylinderDirectionB[5] AND NOT "DB_Outputs".vent[5])));
   "qcylinder6DirectionA" := #_w1;
END_REGION

REGION Network 15: RET CYL 6.- SPARE
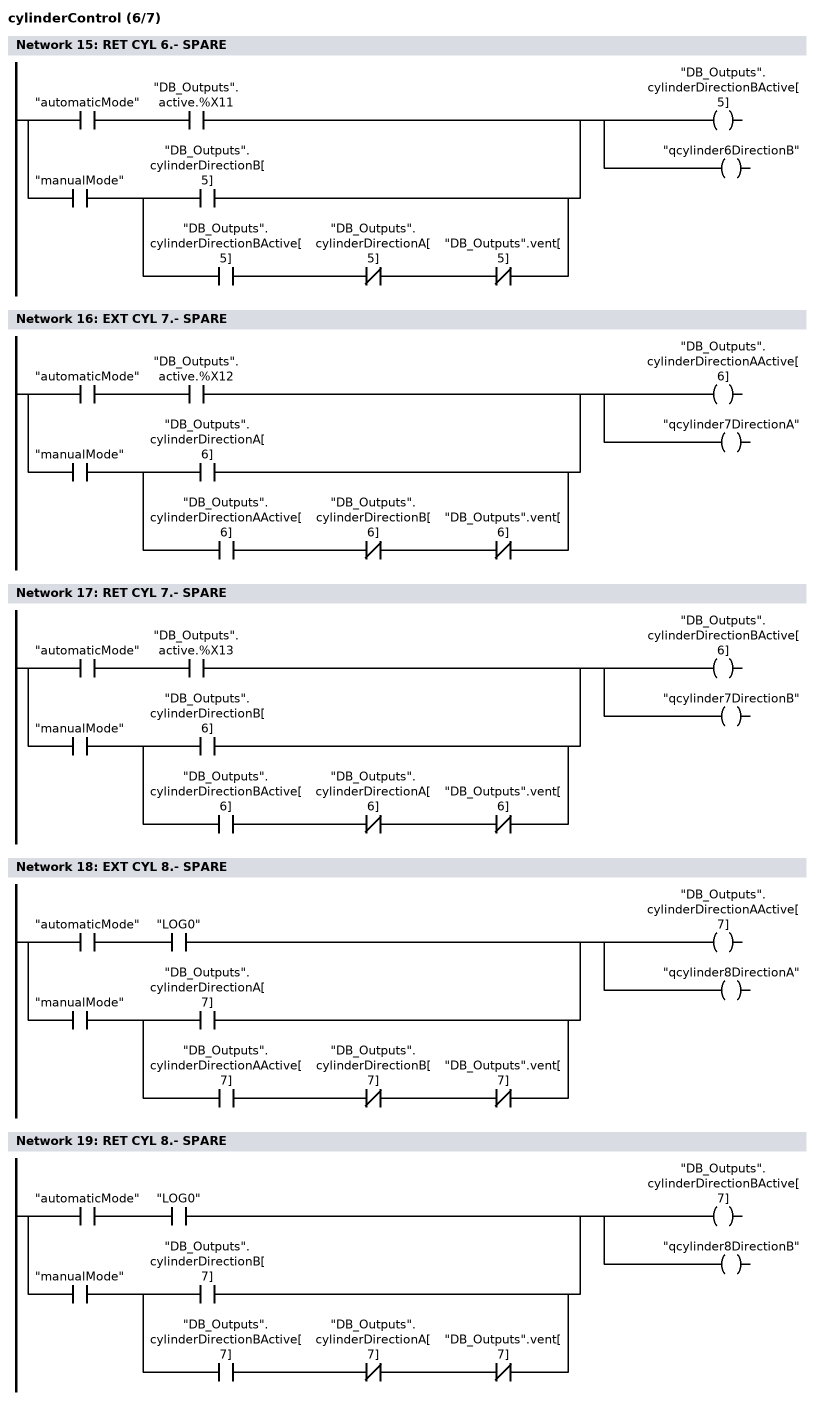
   RUNG wire#powerrail
      Contact( "automaticMode" )
      Contact( "DB_Outputs".active.%X11 )
      wire#w1
      Coil( "DB_Outputs".cylinderDirectionBActive[5] )
   END_RUNG
   RUNG wire#powerrail
      Contact( "manualMode" )
      wire#w2
      Contact( "DB_Outputs".cylinderDirectionB[5] )
   END_RUNG wire#w1
   RUNG wire#w2
      Contact( "DB_Outputs".cylinderDirectionBActive[5] )
      I_Contact( "DB_Outputs".cylinderDirectionA[5] )
      I_Contact( "DB_Outputs".vent[5] )
   END_RUNG wire#w1
   RUNG wire#w1
      Coil( "qcylinder6DirectionB" )
   END_RUNG
   // the same network as SCL:
   #_w1 := ("automaticMode" AND "DB_Outputs".active.%X11) OR ("manualMode" AND ("DB_Outputs".cylinderDirectionB[5] OR ("DB_Outputs".cylinderDirectionBActive[5] AND NOT "DB_Outputs".cylinderDirectionA[5] AND NOT "DB_Outputs".vent[5])));
   "DB_Outputs".cylinderDirectionBActive[5] := ("automaticMode" AND "DB_Outputs".active.%X11) OR ("manualMode" AND ("DB_Outputs".cylinderDirectionB[5] OR ("DB_Outputs".cylinderDirectionBActive[5] AND NOT "DB_Outputs".cylinderDirectionA[5] AND NOT "DB_Outputs".vent[5])));
   "qcylinder6DirectionB" := #_w1;
END_REGION

REGION Network 16: EXT CYL 7.- SPARE
   RUNG wire#powerrail
      Contact( "automaticMode" )
      Contact( "DB_Outputs".active.%X12 )
      wire#w1
      Coil( "DB_Outputs".cylinderDirectionAActive[6] )
   END_RUNG
   RUNG wire#powerrail
      Contact( "manualMode" )
      wire#w2
      Contact( "DB_Outputs".cylinderDirectionA[6] )
   END_RUNG wire#w1
   RUNG wire#w2
      Contact( "DB_Outputs".cylinderDirectionAActive[6] )
      I_Contact( "DB_Outputs".cylinderDirectionB[6] )
      I_Contact( "DB_Outputs".vent[6] )
   END_RUNG wire#w1
   RUNG wire#w1
      Coil( "qcylinder7DirectionA" )
   END_RUNG
   // the same network as SCL:
   #_w1 := ("automaticMode" AND "DB_Outputs".active.%X12) OR ("manualMode" AND ("DB_Outputs".cylinderDirectionA[6] OR ("DB_Outputs".cylinderDirectionAActive[6] AND NOT "DB_Outputs".cylinderDirectionB[6] AND NOT "DB_Outputs".vent[6])));
   "DB_Outputs".cylinderDirectionAActive[6] := ("automaticMode" AND "DB_Outputs".active.%X12) OR ("manualMode" AND ("DB_Outputs".cylinderDirectionA[6] OR ("DB_Outputs".cylinderDirectionAActive[6] AND NOT "DB_Outputs".cylinderDirectionB[6] AND NOT "DB_Outputs".vent[6])));
   "qcylinder7DirectionA" := #_w1;
END_REGION

REGION Network 17: RET CYL 7.- SPARE
   RUNG wire#powerrail
      Contact( "automaticMode" )
      Contact( "DB_Outputs".active.%X13 )
      wire#w1
      Coil( "DB_Outputs".cylinderDirectionBActive[6] )
   END_RUNG
   RUNG wire#powerrail
      Contact( "manualMode" )
      wire#w2
      Contact( "DB_Outputs".cylinderDirectionB[6] )
   END_RUNG wire#w1
   RUNG wire#w2
      Contact( "DB_Outputs".cylinderDirectionBActive[6] )
      I_Contact( "DB_Outputs".cylinderDirectionA[6] )
      I_Contact( "DB_Outputs".vent[6] )
   END_RUNG wire#w1
   RUNG wire#w1
      Coil( "qcylinder7DirectionB" )
   END_RUNG
   // the same network as SCL:
   #_w1 := ("automaticMode" AND "DB_Outputs".active.%X13) OR ("manualMode" AND ("DB_Outputs".cylinderDirectionB[6] OR ("DB_Outputs".cylinderDirectionBActive[6] AND NOT "DB_Outputs".cylinderDirectionA[6] AND NOT "DB_Outputs".vent[6])));
   "DB_Outputs".cylinderDirectionBActive[6] := ("automaticMode" AND "DB_Outputs".active.%X13) OR ("manualMode" AND ("DB_Outputs".cylinderDirectionB[6] OR ("DB_Outputs".cylinderDirectionBActive[6] AND NOT "DB_Outputs".cylinderDirectionA[6] AND NOT "DB_Outputs".vent[6])));
   "qcylinder7DirectionB" := #_w1;
END_REGION

REGION Network 18: EXT CYL 8.- SPARE
   RUNG wire#powerrail
      Contact( "automaticMode" )
      Contact( "LOG0" )
      wire#w1
      Coil( "DB_Outputs".cylinderDirectionAActive[7] )
   END_RUNG
   RUNG wire#powerrail
      Contact( "manualMode" )
      wire#w2
      Contact( "DB_Outputs".cylinderDirectionA[7] )
   END_RUNG wire#w1
   RUNG wire#w2
      Contact( "DB_Outputs".cylinderDirectionAActive[7] )
      I_Contact( "DB_Outputs".cylinderDirectionB[7] )
      I_Contact( "DB_Outputs".vent[7] )
   END_RUNG wire#w1
   RUNG wire#w1
      Coil( "qcylinder8DirectionA" )
   END_RUNG
   // the same network as SCL:
   #_w1 := ("automaticMode" AND "LOG0") OR ("manualMode" AND ("DB_Outputs".cylinderDirectionA[7] OR ("DB_Outputs".cylinderDirectionAActive[7] AND NOT "DB_Outputs".cylinderDirectionB[7] AND NOT "DB_Outputs".vent[7])));
   "DB_Outputs".cylinderDirectionAActive[7] := ("automaticMode" AND "LOG0") OR ("manualMode" AND ("DB_Outputs".cylinderDirectionA[7] OR ("DB_Outputs".cylinderDirectionAActive[7] AND NOT "DB_Outputs".cylinderDirectionB[7] AND NOT "DB_Outputs".vent[7])));
   "qcylinder8DirectionA" := #_w1;
END_REGION

REGION Network 19: RET CYL 8.- SPARE
   RUNG wire#powerrail
      Contact( "automaticMode" )
      Contact( "LOG0" )
      wire#w1
      Coil( "DB_Outputs".cylinderDirectionBActive[7] )
   END_RUNG
   RUNG wire#powerrail
      Contact( "manualMode" )
      wire#w2
      Contact( "DB_Outputs".cylinderDirectionB[7] )
   END_RUNG wire#w1
   RUNG wire#w2
      Contact( "DB_Outputs".cylinderDirectionBActive[7] )
      I_Contact( "DB_Outputs".cylinderDirectionA[7] )
      I_Contact( "DB_Outputs".vent[7] )
   END_RUNG wire#w1
   RUNG wire#w1
      Coil( "qcylinder8DirectionB" )
   END_RUNG
   // the same network as SCL:
   #_w1 := ("automaticMode" AND "LOG0") OR ("manualMode" AND ("DB_Outputs".cylinderDirectionB[7] OR ("DB_Outputs".cylinderDirectionBActive[7] AND NOT "DB_Outputs".cylinderDirectionA[7] AND NOT "DB_Outputs".vent[7])));
   "DB_Outputs".cylinderDirectionBActive[7] := ("automaticMode" AND "LOG0") OR ("manualMode" AND ("DB_Outputs".cylinderDirectionB[7] OR ("DB_Outputs".cylinderDirectionBActive[7] AND NOT "DB_Outputs".cylinderDirectionA[7] AND NOT "DB_Outputs".vent[7])));
   "qcylinder8DirectionB" := #_w1;
END_REGION

REGION Network 20: EXT CYL 9.- SPARE
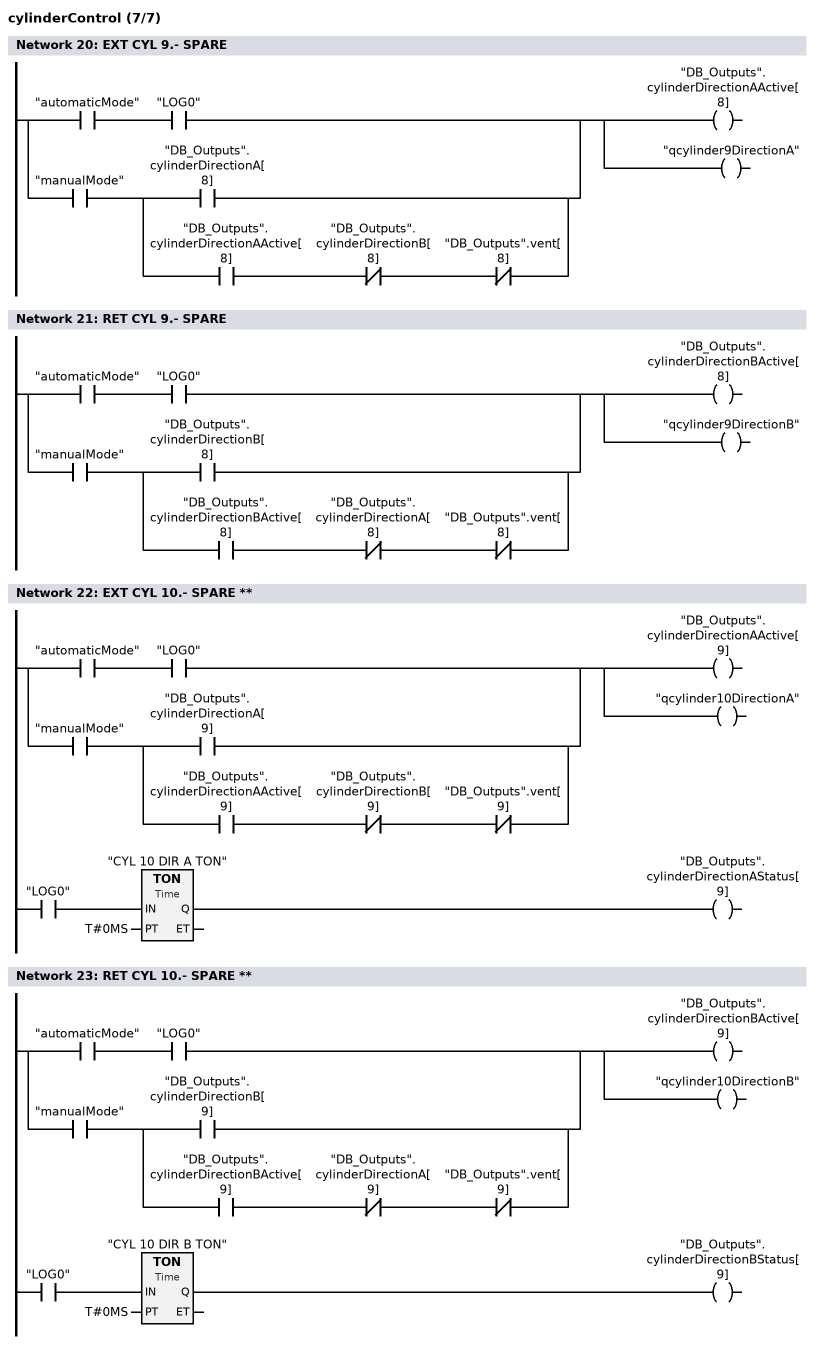
   RUNG wire#powerrail
      Contact( "automaticMode" )
      Contact( "LOG0" )
      wire#w1
      Coil( "DB_Outputs".cylinderDirectionAActive[8] )
   END_RUNG
   RUNG wire#powerrail
      Contact( "manualMode" )
      wire#w2
      Contact( "DB_Outputs".cylinderDirectionA[8] )
   END_RUNG wire#w1
   RUNG wire#w2
      Contact( "DB_Outputs".cylinderDirectionAActive[8] )
      I_Contact( "DB_Outputs".cylinderDirectionB[8] )
      I_Contact( "DB_Outputs".vent[8] )
   END_RUNG wire#w1
   RUNG wire#w1
      Coil( "qcylinder9DirectionA" )
   END_RUNG
   // the same network as SCL:
   #_w1 := ("automaticMode" AND "LOG0") OR ("manualMode" AND ("DB_Outputs".cylinderDirectionA[8] OR ("DB_Outputs".cylinderDirectionAActive[8] AND NOT "DB_Outputs".cylinderDirectionB[8] AND NOT "DB_Outputs".vent[8])));
   "DB_Outputs".cylinderDirectionAActive[8] := ("automaticMode" AND "LOG0") OR ("manualMode" AND ("DB_Outputs".cylinderDirectionA[8] OR ("DB_Outputs".cylinderDirectionAActive[8] AND NOT "DB_Outputs".cylinderDirectionB[8] AND NOT "DB_Outputs".vent[8])));
   "qcylinder9DirectionA" := #_w1;
END_REGION

REGION Network 21: RET CYL 9.- SPARE
   RUNG wire#powerrail
      Contact( "automaticMode" )
      Contact( "LOG0" )
      wire#w1
      Coil( "DB_Outputs".cylinderDirectionBActive[8] )
   END_RUNG
   RUNG wire#powerrail
      Contact( "manualMode" )
      wire#w2
      Contact( "DB_Outputs".cylinderDirectionB[8] )
   END_RUNG wire#w1
   RUNG wire#w2
      Contact( "DB_Outputs".cylinderDirectionBActive[8] )
      I_Contact( "DB_Outputs".cylinderDirectionA[8] )
      I_Contact( "DB_Outputs".vent[8] )
   END_RUNG wire#w1
   RUNG wire#w1
      Coil( "qcylinder9DirectionB" )
   END_RUNG
   // the same network as SCL:
   #_w1 := ("automaticMode" AND "LOG0") OR ("manualMode" AND ("DB_Outputs".cylinderDirectionB[8] OR ("DB_Outputs".cylinderDirectionBActive[8] AND NOT "DB_Outputs".cylinderDirectionA[8] AND NOT "DB_Outputs".vent[8])));
   "DB_Outputs".cylinderDirectionBActive[8] := ("automaticMode" AND "LOG0") OR ("manualMode" AND ("DB_Outputs".cylinderDirectionB[8] OR ("DB_Outputs".cylinderDirectionBActive[8] AND NOT "DB_Outputs".cylinderDirectionA[8] AND NOT "DB_Outputs".vent[8])));
   "qcylinder9DirectionB" := #_w1;
END_REGION

REGION Network 22: EXT CYL 10.- SPARE **
   RUNG wire#powerrail
      Contact( "automaticMode" )
      Contact( "LOG0" )
      wire#w1
      Coil( "DB_Outputs".cylinderDirectionAActive[9] )
   END_RUNG
   RUNG wire#powerrail
      Contact( "manualMode" )
      wire#w2
      Contact( "DB_Outputs".cylinderDirectionA[9] )
   END_RUNG wire#w1
   RUNG wire#w2
      Contact( "DB_Outputs".cylinderDirectionAActive[9] )
      I_Contact( "DB_Outputs".cylinderDirectionB[9] )
      I_Contact( "DB_Outputs".vent[9] )
   END_RUNG wire#w1
   RUNG wire#w1
      Coil( "qcylinder10DirectionA" )
   END_RUNG
   RUNG wire#powerrail
      Contact( "LOG0" )
      { S7_Templates := "time_type := Time" } "CYL 10 DIR A TON".TON(pt := T#0MS, et =>)
      Coil( "DB_Outputs".cylinderDirectionAStatus[9] )
   END_RUNG
   // the same network as SCL:
   #_w1 := ("automaticMode" AND "LOG0") OR ("manualMode" AND ("DB_Outputs".cylinderDirectionA[9] OR ("DB_Outputs".cylinderDirectionAActive[9] AND NOT "DB_Outputs".cylinderDirectionB[9] AND NOT "DB_Outputs".vent[9])));
   "DB_Outputs".cylinderDirectionAActive[9] := ("automaticMode" AND "LOG0") OR ("manualMode" AND ("DB_Outputs".cylinderDirectionA[9] OR ("DB_Outputs".cylinderDirectionAActive[9] AND NOT "DB_Outputs".cylinderDirectionB[9] AND NOT "DB_Outputs".vent[9])));
   "qcylinder10DirectionA" := #_w1;
   "CYL 10 DIR A TON".TON(IN := "LOG0", PT := T#0MS);
   "DB_Outputs".cylinderDirectionAStatus[9] := "CYL 10 DIR A TON".Q;
END_REGION

REGION Network 23: RET CYL 10.- SPARE **
   RUNG wire#powerrail
      Contact( "automaticMode" )
      Contact( "LOG0" )
      wire#w1
      Coil( "DB_Outputs".cylinderDirectionBActive[9] )
   END_RUNG
   RUNG wire#powerrail
      Contact( "manualMode" )
      wire#w2
      Contact( "DB_Outputs".cylinderDirectionB[9] )
   END_RUNG wire#w1
   RUNG wire#w2
      Contact( "DB_Outputs".cylinderDirectionBActive[9] )
      I_Contact( "DB_Outputs".cylinderDirectionA[9] )
      I_Contact( "DB_Outputs".vent[9] )
   END_RUNG wire#w1
   RUNG wire#w1
      Coil( "qcylinder10DirectionB" )
   END_RUNG
   RUNG wire#powerrail
      Contact( "LOG0" )
      { S7_Templates := "time_type := Time" } "CYL 10 DIR B TON".TON(pt := T#0MS, et =>)
      Coil( "DB_Outputs".cylinderDirectionBStatus[9] )
   END_RUNG
   // the same network as SCL:
   #_w1 := ("automaticMode" AND "LOG0") OR ("manualMode" AND ("DB_Outputs".cylinderDirectionB[9] OR ("DB_Outputs".cylinderDirectionBActive[9] AND NOT "DB_Outputs".cylinderDirectionA[9] AND NOT "DB_Outputs".vent[9])));
   "DB_Outputs".cylinderDirectionBActive[9] := ("automaticMode" AND "LOG0") OR ("manualMode" AND ("DB_Outputs".cylinderDirectionB[9] OR ("DB_Outputs".cylinderDirectionBActive[9] AND NOT "DB_Outputs".cylinderDirectionA[9] AND NOT "DB_Outputs".vent[9])));
   "qcylinder10DirectionB" := #_w1;
   "CYL 10 DIR B TON".TON(IN := "LOG0", PT := T#0MS);
   "DB_Outputs".cylinderDirectionBStatus[9] := "CYL 10 DIR B TON".Q;
END_REGION
END_FUNCTION
